Staubli VAL3: cycle_clearList.pgx

program cycle_clearList(num x_nType (dimensions=1))
begin
  logMsg("[KERNEL] PLC:Clear list")
  //
  call processList:deleteAll(x_nType)
end
